# EPICS autosave request: iocBoot/iocPushkar/auto_positions.req
$(P)m1.DVAL
$(P)m2.DVAL
$(P)m3.DVAL
$(P)m4.DVAL
#$(P)m5.DVAL
#$(P)m6.DVAL
#$(P)m7.DVAL
#$(P)m8.DVAL
